FUNCTION_BLOCK FB_ReactorSet_Control
VAR_INPUT
	i_rs_number 			: UINT;
	i_start 				: BOOL;
	i_start_evac			: BOOL;
	i_stop_cmd 				: BOOL;
	i_estop_cmd 			: BOOL;
	i_safe_shutdown			: BOOL;
	i_safe_shutdown_evac 	: BOOL;
	i_reset_fault			: BOOL;
	i_seq_selection			: BYTE;  // 1,2,4,8,16 ( bit 1,2,3,4,5 )
	i_cycles_number			: UINT;
	
	i_cooling_pump_number	: BYTE;
	i_deadair_pump_numner	: BYTE;

	i_adsorption_seq_sts 	: ST_SeqSts;
	i_evac_seq_sts 			: ST_SeqSts;
	i_desorption_seq_sts 	: ST_SeqSts;
	i_cooling_seq_sts 		: ST_SeqSts;
	i_airpress_seq_sts 		: ST_SeqSts;
	
	i_rs_error_active		: BOOL;
	
END_VAR
VAR_OUTPUT
	o_Error 				: BOOL;
	o_Started 				: BOOL;
	o_Done 					: BOOL;
	o_seqStart_req 			: E_RS_SeqState;
	
END_VAR
VAR
	// stateRS :  (Idle := 0,Adsorption := 1,DeadAirEvac := 2,SteamDesorption := 3,VacCooling := 4,AirRepress := 5 , Error := 6);
	seq_state 					: E_RS_SeqState := Idle;
	cycles_to_run 				: UINT;
	cycles_completed			: UINT := 0 ;
	trig_seq_start				: R_TRIG;
	seq_state_first_transition	: BOOL;
	trig_seqstate_first_run		: R_TRIG;
	seq_single_selected			: BOOL;
	
	
END_VAR

CASE seq_state OF 
	
	Idle: 
		 SeqEntry_Handler();
		 trig_seq_start(CLK := i_start) ;
		 IF trig_seq_start.Q THEN 
			 SeqStart_Handler();
			 SeqExit_Handler(i_current_state := Idle);	
		 END_IF
		
	Adsorption :
		SeqEntry_Handler();
		IF NOT i_adsorption_seq_sts.error THEN 	
			IF i_adsorption_seq_sts.completed THEN
				SeqExit_Handler(i_current_state := Adsorption);	
			END_IF
		ELSE
			SeqError_Handler();
		END_IF
	
	DeadAirEvac :
		SeqEntry_Handler();
		IF NOT i_evac_seq_sts.error THEN 	
			IF i_evac_seq_sts.completed THEN
				SeqExit_Handler(i_current_state := DeadAirEvac);	
			END_IF
		ELSE
			SeqError_Handler();
		END_IF
	
	SteamDesorption : 
		SeqEntry_Handler();
		IF NOT i_desorption_seq_sts.error THEN 	
			IF i_desorption_seq_sts.completed THEN
				SeqExit_Handler(i_current_state := SteamDesorption);	
			END_IF
		ELSE
			SeqError_Handler();
		END_IF
	
	VacCooling: 
		SeqEntry_Handler();
		IF NOT i_cooling_seq_sts.error THEN 	
			IF i_cooling_seq_sts.completed THEN
				SeqExit_Handler(i_current_state := VacCooling);	
			END_IF
		ELSE
			SeqError_Handler();
		END_IF
	
	AirRepress :
		SeqEntry_Handler();
		IF NOT i_airpress_seq_sts.error THEN 	
			IF i_airpress_seq_sts.completed THEN
				SeqExit_Handler(i_current_state := AirRepress);			
			END_IF
		ELSE
			SeqError_Handler();
		END_IF
	
	Error : 
		SeqEntry_Handler();
		o_Error := TRUE;
		o_Done := TRUE;
		o_Started := FALSE;
		IF i_reset_fault THEN 
			SeqExit_Handler(i_current_state := Error);	
		END_IF

END_CASE

o_seqStart_req := seq_state;

METHOD Logger : BOOL
VAR_INPUT
END_VAR
ADSLOGSTR(msgCtrlMask := ADSLOG_MSGTYPE_WARN,msgFmtStr := 'Reactor Set : %s' ,strArg := TO_STRING(i_rs_number));
ADSLOGSTR(msgCtrlMask := ADSLOG_MSGTYPE_WARN,msgFmtStr := 'Sequence : %s' ,strArg := TO_STRING(seq_state));
ADSLOGSTR(msgCtrlMask := ADSLOG_MSGTYPE_WARN,msgFmtStr := 'Cycle Number : %s' ,strArg := TO_STRING(cycles_completed));
END_METHOD

METHOD SeqEntry_Handler : BOOL
VAR_INPUT
END_VAR
seq_state_first_transition := TRUE;
trig_seqstate_first_run(CLK := seq_state_first_transition) ;
IF trig_seqstate_first_run.Q THEN 
	Logger();
END_IF
END_METHOD

METHOD SeqError_Handler : BOOL
VAR_INPUT
END_VAR
seq_state_first_transition := FALSE;
trig_seqstate_first_run(CLK := seq_state_first_transition) ;
seq_state := Error;
END_METHOD

METHOD PRIVATE SeqExit_Handler : INT
VAR_INPUT
	i_current_state : E_RS_SeqState;
END_VAR
IF i_current_state = Idle THEN
	o_Done := FALSE;
	o_Started := TRUE;
	o_Error := FALSE;
ELSIF i_stop_cmd OR ((i_current_state = AirRepress) AND (cycles_completed = cycles_to_run)) OR seq_single_selected THEN 
	o_Done := TRUE;
	o_Started := FALSE;
	cycles_completed := 0 ;
	seq_state := Idle;
ELSIF ( i_current_state = AirRepress)  AND ( cycles_completed < cycles_to_run )  THEN 
	seq_state := Adsorption ;
	cycles_completed := cycles_completed + 1;	
ELSIF (NOT ( i_current_state = AirRepress )) AND  (NOT ( i_current_state = Error)) THEN
	seq_state := i_current_state + 1;
ELSIF i_current_state = Error THEN
	o_Error := FALSE;
	seq_state := Idle ;	
END_IF

seq_state_first_transition := FALSE;
trig_seqstate_first_run(CLK := seq_state_first_transition) ;
END_METHOD

METHOD SeqStart_Handler : BOOL
VAR_INPUT
END_VAR
IF i_seq_selection = 0 AND NOT (seq_state = Error) THEN 
	seq_state := Idle;
ELSIF i_seq_selection = 2#11111 THEN
	cycles_to_run := i_cycles_number;
	seq_state_first_transition := FALSE;
	IF i_start_evac THEN 
		seq_state := DeadAirEvac; 
	ELSE
		seq_state := Adsorption;
	END_IF
ELSE
	seq_single_selected := TRUE;	
	seq_state_first_transition := FALSE;
	IF 	i_seq_selection = 2#00001 THEN
		seq_state := Adsorption;
	ELSIF i_seq_selection = 2#00010 THEN
		seq_state := DeadAirEvac;
	ELSIF i_seq_selection = 2#00100 THEN
		seq_state := SteamDesorption;
	ELSIF i_seq_selection = 2#01000 THEN
		seq_state := VacCooling;
	ELSIF i_seq_selection = 2#10000 THEN
		seq_state := AirRepress;
	ELSE
		seq_state := Idle;
	END_IF
END_IF
END_METHOD

PROPERTY SeqState_Sts : E_RS_SeqState
GET
SeqState_Sts := THIS^.seq_state;
END_GET
END_PROPERTY

END_FUNCTION_BLOCK

(* stored: Version 1.1.0.1, ProductVersion 3.1.4024.12
   POU FB_ReactorSet_Control: Id {92b36908-ec7e-40c8-bb48-2c73c6b396cd}, SpecialFunc None
   Method Logger: Id {20227f92-d2b3-4c3b-8917-6409e118b7dd}
   Method SeqEntry_Handler: Id {cd70363c-611b-40f8-a07e-858595aafcb0}
   Method SeqError_Handler: Id {cf16ac2e-ac1f-4245-af07-01d2c1d0d243}
   Method SeqExit_Handler: Id {cf7c1f98-3a99-4ade-b01c-6a2938e0076f}
   Method SeqStart_Handler: Id {5e141aec-f26c-4d41-aa8b-42088dce7405}
   Property SeqState_Sts: Id {ffa55953-79d5-4cd3-a8bf-5e5ae75bb4a3}
   Get Get: Id {5a4664fc-b280-4b10-b244-81551fe54593} *)
